// Uniform read-only view of a device's fault state. Lets aggregator blocks
// (submodule rollups, plant-wide diagnostics) walk a collection of
// unrelated device FBs and query them through a single interface without
// knowing each device's fault enum.
INTERFACE I_Diagnosable

METHOD GetFaultCode : DINT
END_METHOD

METHOD GetFaultString : STRING(79)
END_METHOD

METHOD IsFaulted : BOOL
END_METHOD

END_INTERFACE

(* stored: Version 1.1.0.1, ProductVersion 3.1.4026.12
   Itf I_Diagnosable: Id {b17e48aa-c075-4488-bf95-ed7e41408cdf}
   Method GetFaultCode: Id {c0000005-0000-0000-1000-000000000002}
   Method GetFaultString: Id {c0000005-0000-0000-1000-000000000003}
   Method IsFaulted: Id {97b65ba7-a2c8-4c92-8bf3-4c931f39ad43} *)
